FUNCTION_BLOCK FB_SEL_DT (* F_SEL replacement for DATE_AND_TIME (F_SEL currently doesn't work with DATE_AND_TIME) *)
  (* Standard: 61499-2 *)
  (* Version 1.0, 2017-08-27, Marc Jakobi, HTW Berlin *)
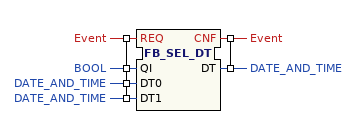
  EVENT_INPUT
    REQ WITH QI, DT0, DT1; (* Normal Execution Request *)
  END_EVENT
  EVENT_OUTPUT
    CNF WITH DT; (* Execution Confirmation *)
  END_EVENT
  VAR_INPUT
    QI : BOOL; (* Input event qualifier *)
    DT0 : DATE_AND_TIME; (* Selectable input variable *)
    DT1 : DATE_AND_TIME; (* Selectable input variable *)
  END_VAR
  VAR_OUTPUT
    DT : DATE_AND_TIME; (* Selected output variable *)
  END_VAR
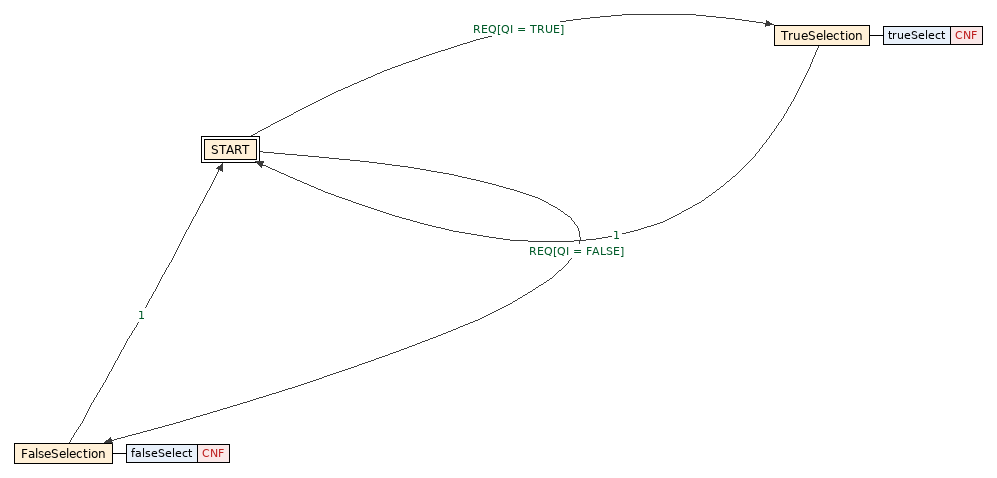
  EC_STATES
    START; (* Initial State *)
    TrueSelection : trueSelect -> CNF; (* Normal execution *)
    FalseSelection : falseSelect -> CNF;
  END_STATES
  EC_TRANSITIONS
    START TO TrueSelection := REQ[QI = TRUE];
    TrueSelection TO START := 1;
    START TO FalseSelection := REQ[QI = FALSE];
    FalseSelection TO START := 1;
  END_TRANSITIONS
  ALGORITHM trueSelect IN ST: (* called upon true input *)
DT :=DT1;
  END_ALGORITHM
  ALGORITHM falseSelect IN ST: (* called upon false input *)
DT := DT0;
  END_ALGORITHM
END_FUNCTION_BLOCK
